FUNCTION_BLOCK D_IN (* Service Interface Function Block Type to ESP32 Module *)
  (* Standard: 61499-2; Description: configurable I/O - INPUT *)
  (* Version 1.0, 2023-12-12, Filipe Gomes *)
  (* Compiler Cpp Unknown Unknown 1.0 *)
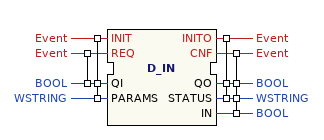
  EVENT_INPUT
    INIT WITH QI, PARAMS; (* Service Initialization *)
    REQ WITH QI; (* Service Request *)
  END_EVENT
  EVENT_OUTPUT
    INITO WITH QO, STATUS; (* Initialization Confirm *)
    CNF WITH QO, STATUS, IN; (* Confirmation of Requested Service *)
  END_EVENT
  VAR_INPUT
    QI : BOOL := TRUE; (* Event Input Qualifier *)
    PARAMS : WSTRING; (* Service Parameters *)
  END_VAR
  VAR_OUTPUT
    QO : BOOL; (* Event Output Qualifier *)
    STATUS : WSTRING; (* Service Status *)
    IN : BOOL; (* Input data from resource *)
  END_VAR
  (* Service /: Service Interface Function Block Type to ESP32 Module *)
END_FUNCTION_BLOCK
